{attribute 'GeneratedUsingTerminal: EL1262-0000-0002'}
{attribute addProperty BoxType "EL1262-0000-0002"}
{attribute addProperty Id "Ch1_CycleCountAT %I*UINT2"}
{attribute addProperty CRC "2646485957"}
{attribute addProperty Size "2"}
TYPE Ch1_CycleCount_9DBE2BC5 :
STRUCT
	{attribute addProperty Name "Ch1_CycleCount"}
	Ch1_CycleCount AT %I* : UINT;
END_STRUCT
END_TYPE

(* stored: Version 1.2.0.0, ProductVersion 3.1.4024.9
   DUT Ch1_CycleCount_9DBE2BC5: Id {c2f8ff8e-e9a6-4b45-93a9-6bde5925e89d} *)
